// NETWORK 4
MC_SetLEPosBias_RightBottom(
    Axis := RightBottomLin,
    ParameterNumber := 1042,
    Value := PositionBias_RightBottom); // MC_WriteParameter

// NETWORK 5
MC_SetLEPosBias_LeftIn(Axis := LeftInLin, ParameterNumber := 1042, Value := PositionBias_LeftIn); // MC_WriteParameter

// NETWORK 6
MC_SetLEPosBias_RightIn(Axis := RightInLin, ParameterNumber := 1042, Value := PositionBias_RightIn); // MC_WriteParameter

// NETWORK 7
MC_SetLEPosBias_LeftOut(Axis := LeftOutLin, ParameterNumber := 1042, Value := PositionBias_LeftOut); // MC_WriteParameter

// NETWORK 8
MC_SetLEPosBias_RightOut(Axis := RightOutLin, ParameterNumber := 1042, Value := PositionBias_RightOut); // MC_WriteParameter
END_ACTION

ACTION A_SetMotorAxisPosition:
fb_ton4_2(PT:=T#0.5S);
CASE SetMotorAxisPosState OF
	0:	(*FB_Set_AxisPosition*)
		FB_Set_MotorAxisPosition(Execute:=TRUE);
		fb_ton4_2.IN:=TRUE;
		SetMotorAxisPosState:=1;
	1:	(*wait*)
		FB_Set_MotorAxisPosition();
		IF NOT FB_Set_MotorAxisPosition.Done THEN		
			IF NOT fb_ton4_2.Q THEN
				SetMotorAxisPosState:=1;
			ELSE
				SetMotorAxisPosState:=99;
			END_IF
		ELSE
			SetMotorAxisPosState:=88;
		END_IF
	88:
		SetMotorAxisPosState:=0;
		SetMotorAxisPositionDone:=TRUE;
		Error:=FALSE;
		ErrorID:=0;
		FB_Set_MotorAxisPosition.Execute:=FALSE;
		fb_ton4_2.IN:=FALSE;
	99:
		SetMotorAxisPosState:=99;
		SetMotorAxisPositionDone:=FALSE;
		Error:=TRUE;
		FB_Set_MotorAxisPosition.Execute:=FALSE;
		fb_ton4_2.IN:=FALSE;
		LED_Error:=TRUE;
		ErrorID:=401;
		ErrorDescription:='SetMotorAxisPosition fail';
END_CASE
END_ACTION

END_PROGRAM
